Fanuc KAREL source: kc00039.KL

-- PROVISIONAL review KL for V1013-1; original PC SHA256 5ed2f0d8b54b4287370edfb0da70c9df23f27ebb7fac587d4e8518f44baac526
-- Incomplete behavior may be omitted. Consult companion uncertainty JSON. Do not deploy.
PROGRAM KC00039
%NOLOCKGROUP
BEGIN
  -- UNRESOLVED_PC offsets 5-32; opcodes 27,22,22,1C,22,76
  -- UNRESOLVED_PC offsets 37-41; opcodes 7F
END KC00039
